Universal Robots PolyScope program: align_for_LtUA.urp

Program align_for_LtUA (installation=default directory=/programs createdIn=5.21.3 lastSavedIn=5.21.3 robotSerialNumber=20246801938)
Calibrated DH parameters: a=[-0.000071, -0.790281, -0.600694, 0.000061, -0.000039, 0]; d=[0.236272, 604.465945, 132.116513, -736.382239, 0.159268, 0.154005]; alpha=[1.570254, -0.000567, 0.000559, 1.571709, -1.56999, 0]; deltaTheta=[0, -0.409357, 7.293326, -0.600784, -0.000001, -0.000001]
InitVariablesNode
Robot Program (runOnlyOnce=true)
  'first move block is unnecessay and bad'
  SuppressedNode
    MoveJ speed 60 deg/s, acceleration 80 deg/s^2 (useActiveTCP=true optimoveEnabled=false optiMoveSpeed=0.3 optiMoveAcceleration=0.09) feature=Base
      'belowis oldhome'
      Waypoint Waypoint_1: TCP in base x=397.354 y=356.263 z=319.809 mm, rx=2.3163 ry=2.0576 rz=0.0741 rad; joints [-198.308, -118.162, 133.452, -12.561, -11.517, -6.326] deg; TCP offset x=-9.5 y=-328 z=105.73 mm, rx=1.2092 ry=-1.2092 rz=1.2092 rad
      SuppressedNode
        Waypoint Waypoint_2: TCP in base x=102.072 y=804.129 z=-21.158 mm, rx=-1.0098 ry=-2.9661 rz=0.0347 rad; joints [-131.791, -72.228, 126.432, -52.794, -4.122, -0.058] deg
      SuppressedNode
        Waypoint Waypoint_3: TCP in base x=-481.576 y=738.776 z=-387.745 mm, rx=-0.0268 ry=3.1371 rz=-0.1325 rad; joints [-88.373, -42.244, 121.849, -79.055, 0.705, 4.289] deg
      Waypoint Waypoint_4: TCP in base x=-790.625 y=220.046 z=-730.503 mm, rx=-0.9425 ry=2.9648 rz=-0.1356 rad; joints [-49.775, -15.59, 117.776, -102.401, 4.996, 5.448] deg
      Waypoint Waypoint_5: TCP in base x=-802.158 y=237.168 z=-730.663 mm, rx=0.8868 ry=-2.4516 rz=0.2829 rad; joints [-61.24, 14.733, 101.407, -222.645, 33.575, 110.967] deg
      Waypoint Waypoint_6: TCP in base x=-687.678 y=589.975 z=-233.622 mm, rx=-0.3444 ry=-1.0001 rz=-2.0808 rad; joints [-61.24, 14.733, 101.407, -222.645, 33.575, -30.853] deg
      SuppressedNode
        Waypoint goalpt: TCP in base x=-796.965 y=229.005 z=-75.004 mm, rx=0 ry=0 rz=-2.526 rad; joints [-49.775, -15.59, 117.776, -102.401, 4.996, -179.788] deg
      Waypoint goalpt2: TCP in base x=-1080.054 y=352.633 z=-86.722 mm, rx=0.0341 ry=-0.0008 rz=-2.631 rad; joints [-41.761, 5.394, 77.547, 101.81, -19.08, -4.137] deg
      Waypoint dummythere: TCP in base x=-1288.589 y=229.005 z=-75.004 mm, rx=0 ry=0 rz=-2.526 rad; joints [-29.748, -12.575, 79.071, -66.58, 25.031, -179.927] deg
  'second one is good'
  SuppressedNode
    MoveJ speed 60 deg/s, acceleration 80 deg/s^2 (useActiveTCP=true optimoveEnabled=false optiMoveSpeed=0.3 optiMoveAcceleration=0.09) feature=Base
      Waypoint goalpt2: TCP in base x=-1080.054 y=352.633 z=-86.722 mm, rx=0.0341 ry=-0.0008 rz=-2.631 rad; joints [-41.761, 5.394, 77.547, 101.81, -19.08, -4.137] deg
  'above was for wrong weldpath'
  SuppressedNode
    Folder savepoints
      MoveJ speed 60 deg/s, acceleration 80 deg/s^2 (useActiveTCP=true optimoveEnabled=false optiMoveSpeed=0.3 optiMoveAcceleration=0.09) feature=Base
        Waypoint leftstart: TCP in base x=-1168.534 y=251.879 z=303.712 mm, rx=-1.4388 ry=-0.6695 rz=0.6003 rad; joints [-161.388, -128.913, -89.606, -145.038, 61.894, 92.57] deg
  SuppressedNode
    MoveJ speed 60 deg/s, acceleration 80 deg/s^2 (useActiveTCP=true optimoveEnabled=false optiMoveSpeed=0.3 optiMoveAcceleration=0.09) feature=Base
      'final point before pa1'
      Waypoint Waypoint_7: TCP in base x=-913.411 y=251.879 z=303.712 mm, rx=-1.2351 ry=-1.1043 rz=1.0523 rad; joints [-156.391, -105.358, -132.178, -128.187, 33.298, 95.672] deg
      'oldhome'
      Waypoint Waypoint_8: TCP in base x=397.354 y=356.263 z=319.809 mm, rx=2.3163 ry=2.0576 rz=0.0741 rad; joints [-198.308, -118.162, 133.452, -12.561, -11.517, -6.326] deg
  MoveJ speed 60 deg/s, acceleration 80 deg/s^2 (useActiveTCP=true optimoveEnabled=false optiMoveSpeed=0.3 optiMoveAcceleration=0.09) feature=Base
    'from oldhome, actual path'
    SuppressedNode
      Waypoint Waypoint_9: TCP in base x=683.137 y=304.628 z=775.294 mm, rx=1.9572 ry=1.7212 rz=0.4516 rad; joints [-193.46, -116.682, 102.732, -25.933, -6.334, 5.47] deg
    SuppressedNode
      Waypoint Waypoint_10: TCP in base x=-197.847 y=491.143 z=1723.576 mm, rx=-0.0125 ry=0.2444 rz=1.7982 rad; joints [-175.692, -50.406, -94.795, -74.947, 12.663, 48.707] deg
    Waypoint Waypoint_13: TCP in base x=-814.246 y=233.556 z=311.707 mm, rx=0.0475 ry=0.0091 rz=-2.8285 rad; joints [-48.272, -48.097, 133.86, -81.091, 23.95, 175.661] deg
    SuppressedNode
      Waypoint Waypoint_12: TCP in base x=-793.876 y=251.879 z=303.712 mm, rx=-1.2351 ry=-1.1043 rz=1.0523 rad; joints [-150.736, -98.884, -141.754, -124.357, 38.932, 94.772] deg
  SuppressedNode
    MoveJ speed 60 deg/s, acceleration 80 deg/s^2 (useActiveTCP=true optimoveEnabled=false optiMoveSpeed=0.3 optiMoveAcceleration=0.09) feature=Base
      SuppressedNode
        Waypoint Waypoint_12: TCP in base x=-793.876 y=251.879 z=303.712 mm, rx=-1.2351 ry=-1.1043 rz=1.0523 rad; joints [-150.736, -98.884, -141.754, -124.357, 38.932, 94.772] deg
      Waypoint Waypoint_28: TCP in base x=-612.422 y=86.102 z=307.954 mm, rx=0.0596 ry=0.0051 rz=-1.7683 rad; joints [-50.054, -48.046, 134.598, -90.438, -38.763, -175.268] deg
  SuppressedNode
    Folder dummy points
      'for seeing if it goes to each side correctly'
      MoveJ speed 60 deg/s, acceleration 80 deg/s^2 (useActiveTCP=true optimoveEnabled=false optiMoveSpeed=0.3 optiMoveAcceleration=0.09) feature=Base
        'right side weld'
        Waypoint Waypoint_15: TCP in base x=-1072.479 y=376.012 z=295.965 mm, rx=-0.7812 ry=-1.774 rz=1.7129 rad; joints [-196.962, -109.785, -121.389, -129.338, -59.875, 88.022] deg
      MoveL speed 10 mm/s, acceleration 50 mm/s^2 (useActiveTCP=true optimoveEnabled=false optiMoveSpeed=0.3 optiMoveAcceleration=0.09) feature=Base
        Waypoint Waypoint_14: TCP in base x=-1156.816 y=297.468 z=291.375 mm, rx=-0.7812 ry=-1.774 rz=1.7129 rad; joints [-189.786, -111.954, -118.346, -130.254, -52.7, 88.101] deg
      MoveJ speed 60 deg/s, acceleration 80 deg/s^2 (useActiveTCP=true optimoveEnabled=false optiMoveSpeed=0.3 optiMoveAcceleration=0.09) feature=Base
        Waypoint Waypoint_16: TCP in base x=-632.457 y=-64.235 z=338.109 mm, rx=-1.488 ry=-0.4247 rz=0.3419 rad; joints [-132.464, -114.908, -114.428, -134.512, 109.372, 90.647] deg; TCP offset x=4.51 y=-328 z=105.73 mm, rx=1.2092 ry=-1.2092 rz=1.2092 rad
      MoveJ speed 60 deg/s, acceleration 80 deg/s^2 (useActiveTCP=true optimoveEnabled=false optiMoveSpeed=0.3 optiMoveAcceleration=0.09) feature=Base
        'ltua'
        Waypoint Waypoint_17: TCP in base x=-1093.81 y=272.866 z=328.409 mm, rx=-0.0256 ry=0.0599 rz=-2.4904 rad; joints [-37.936, -41.228, 103.516, -63.348, 14.845, -181.804] deg; TCP offset x=-9.5 y=-328 z=105.73 mm, rx=1.2092 ry=-1.2092 rz=1.2092 rad
        Waypoint Waypoint_18: TCP in base x=-1061.025 y=229.781 z=325.732 mm, rx=-0.0256 ry=0.0599 rz=-2.4904 rad; joints [-37.091, -42.558, 107.981, -66.424, 15.69, -181.866] deg
        Waypoint Waypoint_19: TCP in base x=-1061.025 y=229.781 z=325.732 mm, rx=-0.0004 ry=-0.074 rz=2.9743 rad; joints [-28.832, -45.944, 119.574, -73.914, 70.757, -182.737] deg
        Waypoint Waypoint_20: TCP in base x=-1061.025 y=229.781 z=325.732 mm, rx=-0.0238 ry=-0.0561 rz=2.18 rad; joints [-15.091, -44.425, 114.036, -69.96, 130.027, -183.054] deg
        Waypoint Waypoint_21: TCP in base x=-1140.96 y=164.286 z=320.912 mm, rx=-0.0238 ry=-0.0561 rz=2.18 rad; joints [-9.977, -41.867, 106.747, -65.258, 135.141, -183.096] deg
        Waypoint Waypoint_22: TCP in base x=-1053.643 y=226.515 z=320.912 mm, rx=-0.0251 ry=0.0605 rz=-2.5121 rad; joints [-37.141, -42.631, 109.143, -67.442, 16.887, -181.94] deg
        Waypoint Waypoint_23: TCP in base x=-1028.819 y=192.377 z=318.826 mm, rx=-0.0251 ry=0.0605 rz=-2.5121 rad; joints [-36.351, -43.503, 112.437, -69.82, 17.677, -181.985] deg
        Waypoint Waypoint_24: TCP in base x=-1028.819 y=192.377 z=318.826 mm, rx=0.3097 ry=-0.9677 rz=-2.3496 rad; joints [-29.857, -55.018, 130.517, -76.163, 24.172, -134.695] deg
        Waypoint Waypoint_25: TCP in base x=-1028.819 y=192.377 z=318.826 mm, rx=0.5985 ry=-1.8525 rz=-1.8653 rad; joints [-25.796, -76.67, 133.521, -57.465, 28.235, -89.911] deg
        Waypoint Waypoint_26: TCP in base x=-1025.481 y=190.565 z=741.7 mm, rx=0.5985 ry=-1.8525 rz=-1.8653 rad; joints [-25.76, -97.088, 113.302, -16.887, 28.26, -89.844] deg
      MoveJ speed 60 deg/s, acceleration 80 deg/s^2 (useActiveTCP=true optimoveEnabled=false optiMoveSpeed=0.3 optiMoveAcceleration=0.09) feature=Base
        Waypoint Waypoint_27: TCP in base x=-793.23 y=192.377 z=318.826 mm, rx=-0.0064 ry=0.0033 rz=-2.5127 rad; joints [-47.834, -47.702, 132.041, -86.771, 6.192, -177.807] deg
        Waypoint Waypoint_28: TCP in base x=-612.422 y=86.102 z=307.954 mm, rx=0.0596 ry=0.0051 rz=-1.7683 rad; joints [-50.054, -48.046, 134.598, -90.438, -38.763, -175.268] deg
        Waypoint Waypoint_29: TCP in base x=445.167 y=807.566 z=370.842 mm, rx=0.9155 ry=2.0728 rz=1.7665 rad; joints [-158.883, -80.173, 129.572, -27.753, -31.851, -95.578] deg
      MoveJ speed 60 deg/s, acceleration 80 deg/s^2 (useActiveTCP=true optimoveEnabled=false optiMoveSpeed=0.3 optiMoveAcceleration=0.09) feature=Base
        'actual '
        Waypoint Waypoint_11: TCP in base x=-1049.666 y=233.556 z=311.707 mm, rx=-0.0387 ry=0.0168 rz=2.2542 rad; joints [-15.283, -44.427, 115.215, -68.464, 125.588, 181.289] deg
        Waypoint Waypoint_13: TCP in base x=-814.246 y=233.556 z=311.707 mm, rx=0.0475 ry=0.0091 rz=-2.8285 rad; joints [-48.272, -48.097, 133.86, -81.091, 23.95, 175.661] deg
